FUNCTION_BLOCK xaxpy_dmyzr5
VAR_INPUT
    b_n: DINT;
    a: LREAL;
    x: ARRAY [0..5] OF LREAL;
    ix0: DINT;
    iy0: DINT;
END_VAR
VAR_IN_OUT
    y: ARRAY [0..35] OF LREAL;
END_VAR
VAR_TEMP
    ix: DINT;
    iy: DINT;
    k: DINT;
END_VAR

IF (b_n >= 1) AND (a <> 0.0) THEN 
    ix := ix0 - 1;
    iy := iy0 - 1;
    k := 0;
    WHILE k <= (b_n - 1) DO
        y[iy] := (a * x[ix]) + y[iy];
        ix := ix + 1;
        iy := iy + 1;
        k := k + 1;
    END_WHILE;
END_IF;

END_FUNCTION_BLOCK

(* stored: Version 1.1.0.1, ProductVersion 3.1.4024.12
   POU xaxpy_dmyzr5: Id {04db2957-c03b-4c68-b155-509de2b774ce}, SpecialFunc None *)
